{attribute 'qualified_only'}
{attribute 'strict'}
{attribute 'to_string'}
TYPE eTcaWorkpiecePlaceStatus :
(
	undefined := 0,
	Ready,
	Prepared,
	Loaded,	
	Locked,
	
	MAXSIZE
);
END_TYPE

(* stored: Version 1.1.0.1
   DUT eTcaWorkpiecePlaceStatus: Id {d29c626f-62d9-4d08-87c8-1233417dc64f} *)
